PROGRAM Move_JOG
VAR
	
END_VAR

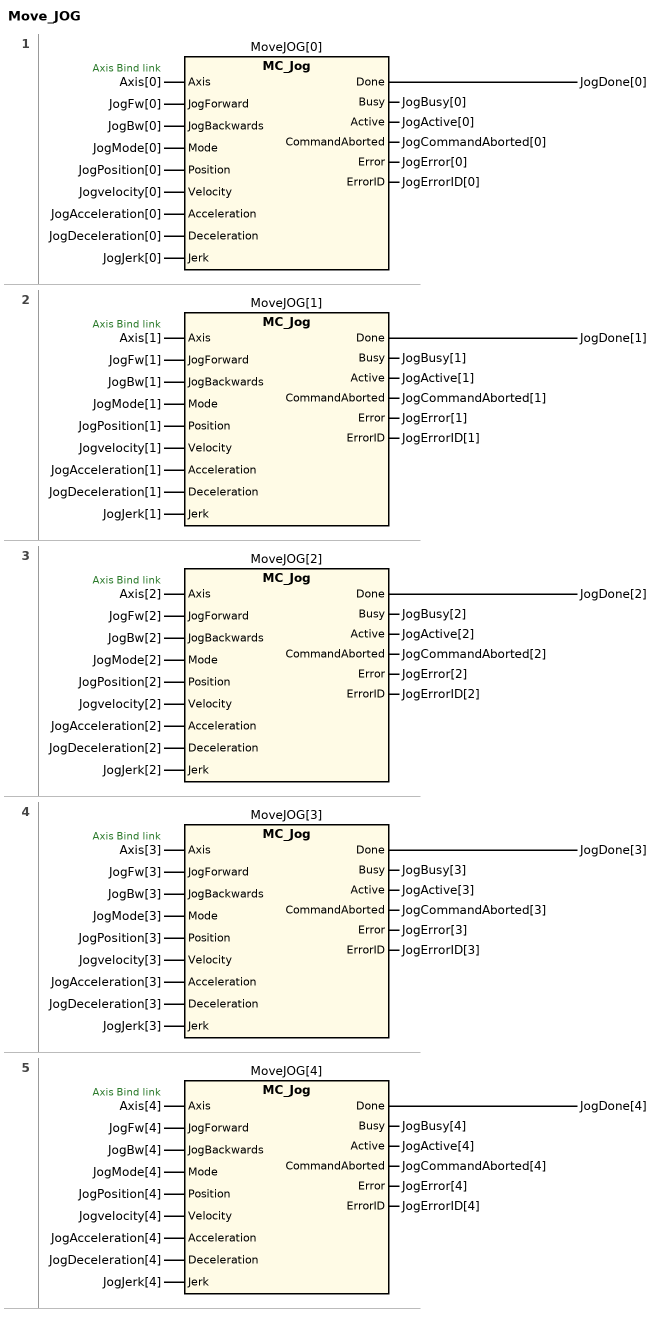
// NETWORK 1
//   MoveJOG[0]: MoveJOG
//   Axis[0]: Axis Bind link
MoveJOG[0](
    Axis := Axis[0],
    JogForward := JogFw[0],
    JogBackwards := JogBw[0],
    Mode := JogMode[0],
    Position := JogPosition[0],
    Velocity := Jogvelocity[0],
    Acceleration := JogAcceleration[0],
    Deceleration := JogDeceleration[0],
    Jerk := JogJerk[0],
    Busy => JogBusy[0],
    Active => JogActive[0],
    CommandAborted => JogCommandAborted[0],
    Error => JogError[0],
    ErrorID => JogErrorID[0]); // MC_Jog
JogDone[0] := MoveJOG[0].Done;

// NETWORK 2
//   MoveJOG[1]: MoveJOG
//   Axis[1]: Axis Bind link
MoveJOG[1](
    Axis := Axis[1],
    JogForward := JogFw[1],
    JogBackwards := JogBw[1],
    Mode := JogMode[1],
    Position := JogPosition[1],
    Velocity := Jogvelocity[1],
    Acceleration := JogAcceleration[1],
    Deceleration := JogDeceleration[1],
    Jerk := JogJerk[1],
    Busy => JogBusy[1],
    Active => JogActive[1],
    CommandAborted => JogCommandAborted[1],
    Error => JogError[1],
    ErrorID => JogErrorID[1]); // MC_Jog
JogDone[1] := MoveJOG[1].Done;

// NETWORK 3
//   MoveJOG[2]: MoveJOG
//   Axis[2]: Axis Bind link
MoveJOG[2](
    Axis := Axis[2],
    JogForward := JogFw[2],
    JogBackwards := JogBw[2],
    Mode := JogMode[2],
    Position := JogPosition[2],
    Velocity := Jogvelocity[2],
    Acceleration := JogAcceleration[2],
    Deceleration := JogDeceleration[2],
    Jerk := JogJerk[2],
    Busy => JogBusy[2],
    Active => JogActive[2],
    CommandAborted => JogCommandAborted[2],
    Error => JogError[2],
    ErrorID => JogErrorID[2]); // MC_Jog
JogDone[2] := MoveJOG[2].Done;

// NETWORK 4
//   MoveJOG[3]: MoveJOG
//   Axis[3]: Axis Bind link
MoveJOG[3](
    Axis := Axis[3],
    JogForward := JogFw[3],
    JogBackwards := JogBw[3],
    Mode := JogMode[3],
    Position := JogPosition[3],
    Velocity := Jogvelocity[3],
    Acceleration := JogAcceleration[3],
    Deceleration := JogDeceleration[3],
    Jerk := JogJerk[3],
    Busy => JogBusy[3],
    Active => JogActive[3],
    CommandAborted => JogCommandAborted[3],
    Error => JogError[3],
    ErrorID => JogErrorID[3]); // MC_Jog
JogDone[3] := MoveJOG[3].Done;

// NETWORK 5
//   MoveJOG[4]: MoveJOG
//   Axis[4]: Axis Bind link
MoveJOG[4](
    Axis := Axis[4],
    JogForward := JogFw[4],
    JogBackwards := JogBw[4],
    Mode := JogMode[4],
    Position := JogPosition[4],
    Velocity := Jogvelocity[4],
    Acceleration := JogAcceleration[4],
    Deceleration := JogDeceleration[4],
    Jerk := JogJerk[4],
    Busy => JogBusy[4],
    Active => JogActive[4],
    CommandAborted => JogCommandAborted[4],
    Error => JogError[4],
    ErrorID => JogErrorID[4]); // MC_Jog
JogDone[4] := MoveJOG[4].Done;

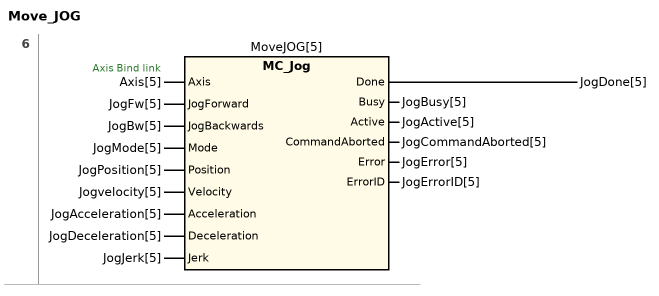
// NETWORK 6
//   MoveJOG[5]: MoveJOG
//   Axis[5]: Axis Bind link
MoveJOG[5](
    Axis := Axis[5],
    JogForward := JogFw[5],
    JogBackwards := JogBw[5],
    Mode := JogMode[5],
    Position := JogPosition[5],
    Velocity := Jogvelocity[5],
    Acceleration := JogAcceleration[5],
    Deceleration := JogDeceleration[5],
    Jerk := JogJerk[5],
    Busy => JogBusy[5],
    Active => JogActive[5],
    CommandAborted => JogCommandAborted[5],
    Error => JogError[5],
    ErrorID => JogErrorID[5]); // MC_Jog
JogDone[5] := MoveJOG[5].Done;

END_PROGRAM

(* stored: Version 1.1.0.1, ProductVersion 3.1.4018.5
   POU Move_JOG: Id {158d760c-74ba-43c1-a5d8-a9e10dcd9a96}, SpecialFunc None *)
